FUNCTION_BLOCK Multiplexer
VAR_INPUT
	In1: BOOL;
	In2: BOOL;
	In4: BOOL;
	In3: BOOL;
END_VAR

VAR_OUTPUT
	Out1: BOOL;
	Out2: BOOL;
	Out3: BOOL;
	Out4: BOOL;
END_VAR

VAR
	UpDown: RS;
	CWCCW: RS;
	StretchShrink: RS;
	GrabRelease: RS;
END_VAR

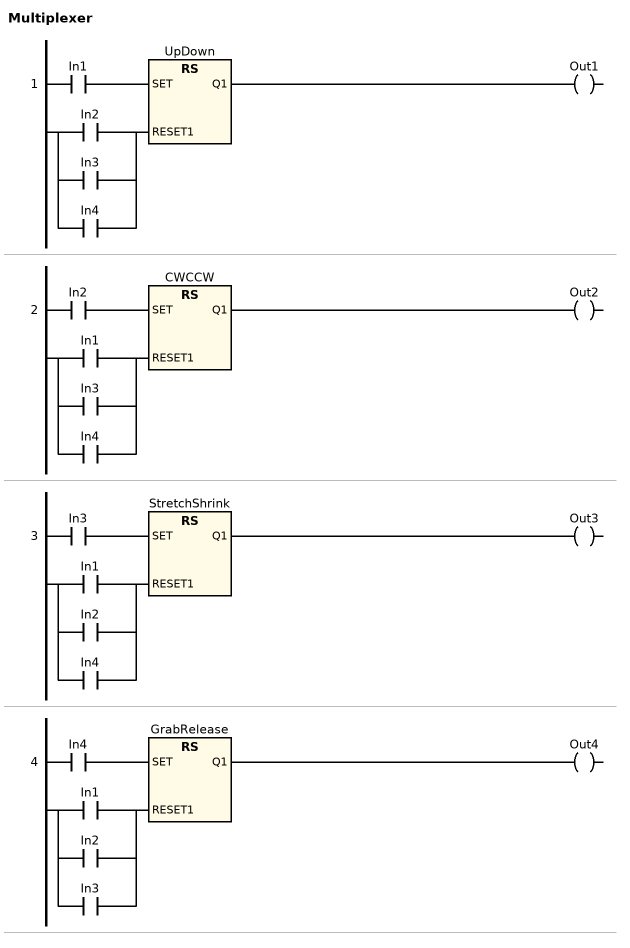
// NETWORK 1
UpDown(SET := In1, RESET1 := In2 OR In3 OR In4); // RS
Out1 := UpDown.Q1;

// NETWORK 2
CWCCW(SET := In2, RESET1 := In1 OR In3 OR In4); // RS
Out2 := CWCCW.Q1;

// NETWORK 3
StretchShrink(SET := In3, RESET1 := In1 OR In2 OR In4); // RS
Out3 := StretchShrink.Q1;

// NETWORK 4
GrabRelease(SET := In4, RESET1 := In1 OR In2 OR In3); // RS
Out4 := GrabRelease.Q1;

END_FUNCTION_BLOCK

(* stored: Version 1.1.0.1, ProductVersion 3.1.4024.15
   POU Multiplexer: Id {7dee7065-95cf-476e-aef2-4cc3b00f1a1f}, SpecialFunc None *)
